{attribute 'linkalways'} 
{attribute 'no_explicit_call' := 'This FB is a CLASS and must be accessed using methods or properties'}
{attribute 'enable_dynamic_creation'}
FUNCTION_BLOCK FINAL ADD_SINT EXTENDS Node
VAR
	in1 : _SINT(0);
	in2 : _SINT(0);
	out : _SINT(0);
END_VAR

METHOD PUBLIC Clone : I_Node
VAR
	pNode : POINTER TO ADD_SINT;
END_VAR
pNode := __NEW(ADD_SINT);
Clone := pNode^;
END_METHOD

METHOD FB_init : BOOL
VAR_INPUT
	bInitRetains : BOOL; // if TRUE, the retain variables are initialized (warm start / cold start)
	bInCopyCode : BOOL;  // if TRUE, the instance afterwards gets moved into the copy code (online change)
END_VAR
AddInput('in1',THIS^.in1);
AddInput('in2',THIS^.in2);
AddOutput('out', THIS^.out);
END_METHOD

METHOD PROTECTED OnExecute
VAR
END_VAR
out.Value := in1.Value + in2.Value;
END_METHOD

END_FUNCTION_BLOCK

(* stored: Version 1.1.0.1, ProductVersion 3.1.4024.15
   POU ADD_SINT: Id {317b749b-a3f5-4fa9-98c2-ce2ced2e7bc0}, SpecialFunc None
   Folder Constructor: Id {f31168e4-466a-41ae-9258-73521355a18b}
   Method Clone: Id {b1f8b6f4-8e6b-487d-8931-6f56d2931e7e}
   Method FB_init: Id {84c1cce0-f2f2-417d-84be-168b23bba0f1}
   Method OnExecute: Id {a3ac6b40-db5c-4baa-9018-786bb90dbde7} *)
